// TIA Portal project "Delayed Motor Start and Pump Control via Pushbutton in Siemens PLC" (V17)
// Delayed Motor Start and Pump Control via Pushbutton in Siemens PLC
// When Start Pushbutton is pressed and released, then Motor will be ON after 15 sec.
// When Stop Pushbutton is pressed and released, then Motor will stop immediately and Pump will turn ON after 10 sec.

(* hardware
DEVICE "S7-1200 station_1"  S7-1200 Station
   slot 0: "Rack_0"  S7-1200 Rack  Rack  V1.0
   slot 1: "PLC_1"  CPU 1212C DC/DC/DC  6ES7 212-1AE40-0XB0  V4.5
*)

// ===== PLC "PLC_1"  CPU 1212C DC/DC/DC =====

VAR_GLOBAL   // PLC tag table "Default tag table"
   "Start pushbutton" AT %I0.0 : Bool;
   "Stop pushbutton" AT %I0.1 : Bool;
   "Motor" AT %Q0.0 : Bool;
   "Pump" AT %Q0.1 : Bool;
   "Tag_1" AT %M0.0 : Bool;
   "Tag_2" AT %M0.1 : Bool;
END_VAR

// folder: System blocks/Program resources

DATA_BLOCK "IEC_Timer_0_DB"   // DB1
{ S7_Optimized_Access := 'TRUE' }
AUTHOR : Simatic
FAMILY : IEC
NAME : IEC_TMR
VERSION : 1.0
// stored: InstanceOfName IEC_TIMER
"IEC_TIMER"
BEGIN
END_DATA_BLOCK

DATA_BLOCK "IEC_Timer_0_DB_1"   // DB2
{ S7_Optimized_Access := 'TRUE' }
AUTHOR : Simatic
FAMILY : IEC
NAME : IEC_TMR
VERSION : 1.0
// stored: InstanceOfName IEC_TIMER
"IEC_TIMER"
BEGIN
END_DATA_BLOCK

// folder: (top level)

ORGANIZATION_BLOCK "Main"   // OB1, LAD, ProgramCycle
TITLE = "Main Program Sweep (Cycle)"
{ S7_Optimized_Access := 'TRUE' }
VERSION : 0.1
   VAR_INPUT
      Initial_Call : Bool;   // Initial call of this OB
      Remanence : Bool;   // =True, if remanent data are available
   END_VAR
BEGIN

REGION Network 1
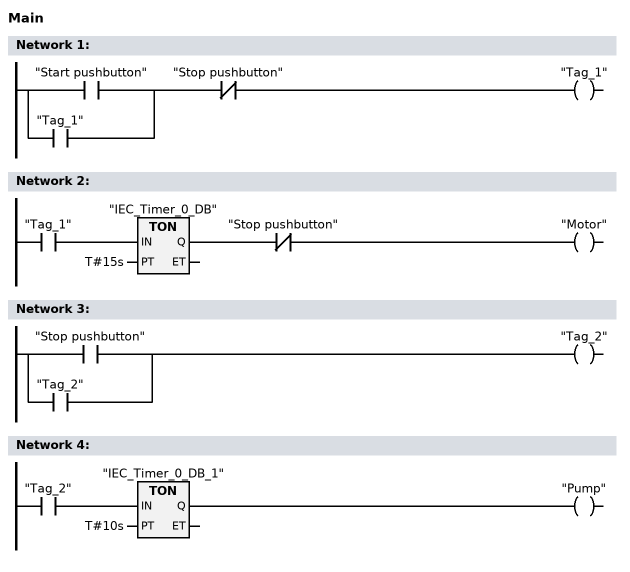
   RUNG wire#powerrail
      Contact( "Start pushbutton" )
      wire#w1
      I_Contact( "Stop pushbutton" )
      Coil( "Tag_1" )
   END_RUNG
   RUNG wire#powerrail
      Contact( "Tag_1" )
   END_RUNG wire#w1
   // the same network as SCL:
   "Tag_1" := ("Start pushbutton" OR "Tag_1") AND NOT "Stop pushbutton";
END_REGION

REGION Network 2
   "IEC_Timer_0_DB".TON(IN := "Tag_1", PT := T#15s);
   "Motor" := "IEC_Timer_0_DB".Q AND NOT "Stop pushbutton";
END_REGION

REGION Network 3
   RUNG wire#powerrail
      Contact( "Stop pushbutton" )
      wire#w1
      Coil( "Tag_2" )
   END_RUNG
   RUNG wire#powerrail
      Contact( "Tag_2" )
   END_RUNG wire#w1
   // the same network as SCL:
   "Tag_2" := "Stop pushbutton" OR "Tag_2";
END_REGION

REGION Network 4
   "IEC_Timer_0_DB_1".TON(IN := "Tag_2", PT := T#10s);
   "Pump" := "IEC_Timer_0_DB_1".Q;
END_REGION
END_ORGANIZATION_BLOCK